TYPE ST_ClosedLoopControlSettings :
STRUCT
	fMaxPositionError 					: LREAL;
	fProportionalGain 					: LREAL;
	fIntegralGain 						: LREAL;
END_STRUCT
END_TYPE

(* stored: Version 1.1.0.1, ProductVersion 3.1.4024.11
   DUT ST_ClosedLoopControlSettings: Id {7ee854d9-b6f8-4d51-b179-a1136b0ccbb8} *)
